{attribute 'qualified_only'}
VAR_GLOBAL CONSTANT
	DefaultSensorElement : E_Mfr_MeasuringElement := E_Mfr_MeasuringElement.eNI1000;
END_VAR

(* stored: Version 1.1.0.1
   GVL Mfr_Param: Id {51355aa6-818b-4990-900f-53c437098ad2}, ParameterList True *)
